{attribute 'GeneratedUsingTerminal: EK1100-0000-0018'}
{attribute addProperty BoxType "EK1100-0000-0018"}
{attribute addProperty Id "Beckhoff_EL19xxEK1122Beckhoff_EL19xxEK1122_2AE5B5792A_0001_EL1918_0000_0016EL1918_414C842648"}
{attribute addProperty CRC "3377794039"}
{attribute addProperty Size "50"}
TYPE Beckhoff_EL19xx_C9550BF7 EXTENDS EK1100_1FC0878B :
STRUCT
	{attribute addProperty Name "Beckhoff_EL19xxEK1122"}
	{attribute addProperty PreviousPort "Beckhoff EL19xx : B"}
	Beckhoff_EL19xxEK1122 : Beckhoff_EL19xxEK1122_2AE5B579;
	{attribute addProperty Name "A_0001_EL1918_0000_0016"}
	{attribute addProperty PreviousPort "Beckhoff EL19xxEK1122 : C"}
	A_0001_EL1918_0000_0016 : EL1918_414C8426;
END_STRUCT
END_TYPE

(* stored: Version 1.2.0.0, ProductVersion 3.1.4024.9
   DUT Beckhoff_EL19xx_C9550BF7: Id {2b08e4f9-7719-49f1-b434-ffeb4c31de78} *)
